FUNCTION TryConvert_UDINT_TO_DT : BOOL
VAR_INPUT
	in : UDINT;
	out : REFERENCE TO DT;
END_VAR

out := UDINT_TO_DT(in);
TryConvert_UDINT_TO_DT := TRUE;

END_FUNCTION

(* stored: Version 1.1.0.1, ProductVersion 3.1.4024.12
   POU TryConvert_UDINT_TO_DT: Id {a7abb6ed-7ec6-431b-9712-2c6ebbcd449a}, SpecialFunc None *)
